# EPICS autosave request: iocs/ADCrayDlIOC/iocBoot/iocRayonix/auto_settings.req
file "ADCrayDl_settings.req",    P=$(P),  R=cam1:
file "NDStdArrays_settings.req",    P=$(P),  R=image1:
